Universal Robots PolyScope program: programa3.urp

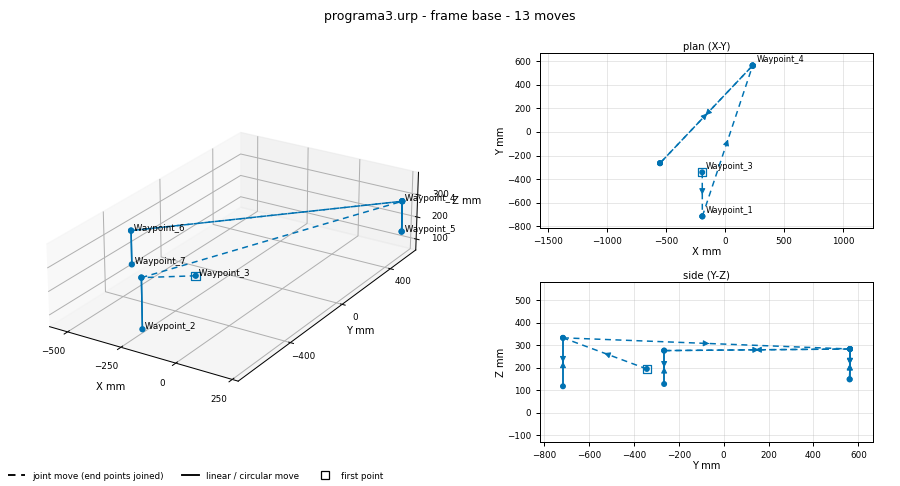
[picture p0: tool path of programa3.urp in frame base, 13 of 13 moves have a stored position in this frame; points joined in program order, loops and branches not executed]
Program programa3 (installation=default directory=/ursim/programs createdIn=5.26.1 lastSavedIn=5.26.1 robotSerialNumber=20195599999)
Calibrated DH parameters: a=[0, -0.425, -0.3922, 0, 0, 0]; d=[0.1625, 0, 0, 0.1333, 0.0997, 0.0996]; alpha=[1.570796, 0, 0, 1.570796, -1.570796, 0]; deltaTheta=[0, 0, 0, 0, 0, 0]
InitVariablesNode
Robot Program (runOnlyOnce=false)
  MoveJ speed 60 deg/s, acceleration 80 deg/s^2 (useActiveTCP=true optimoveEnabled=false optiMoveSpeed=0.3 optiMoveAcceleration=0.09) feature=Base
    Waypoint Waypoint_3: TCP in base x=-191.294 y=-341.962 z=194.296 mm, rx=-0.0012 ry=3.1163 rz=0.0389 rad; joints [-99.651, -91.23, -136.603, -43.818, 91.176, -9.713] deg; TCP offset x=0 y=0 z=0 mm, rx=0 ry=0 rz=0 rad
  Loop Forever
    MoveJ speed 60 deg/s, acceleration 80 deg/s^2 (useActiveTCP=true optimoveEnabled=false optiMoveSpeed=0.3 optiMoveAcceleration=0.09) feature=Base
      Waypoint Waypoint_1: TCP in base x=-190.469 y=-715.405 z=332.843 mm, rx=-0.0012 ry=3.1163 rz=0.0389 rad; joints [-94.715, -125.441, -65.388, -80.715, 91.313, -4.778] deg; TCP offset x=0 y=0 z=0 mm, rx=0 ry=0 rz=0 rad
    MoveL speed 250 mm/s, acceleration 1200 mm/s^2 (useActiveTCP=true optimoveEnabled=false optiMoveSpeed=0.3 optiMoveAcceleration=0.09) feature=Base
      Waypoint Waypoint_2: TCP in base x=-190.469 y=-715.405 z=116.996 mm, rx=-0.0012 ry=3.1163 rz=0.0389 rad; joints [-94.715, -137.604, -78.272, -55.669, 91.313, -4.778] deg; TCP offset x=0 y=0 z=0 mm, rx=0 ry=0 rz=0 rad
    Set DigitalOutput pin=digital_out[0]; digitalValue=1
    Wait Sleep waitTime=1
    MoveL speed 250 mm/s, acceleration 1200 mm/s^2 (useActiveTCP=true optimoveEnabled=false optiMoveSpeed=0.3 optiMoveAcceleration=0.09) feature=Base
      Waypoint Waypoint_1: TCP in base x=-190.469 y=-715.405 z=332.843 mm, rx=-0.0012 ry=3.1163 rz=0.0389 rad; joints [-94.715, -125.441, -65.388, -80.715, 91.313, -4.778] deg; TCP offset x=0 y=0 z=0 mm, rx=0 ry=0 rz=0 rad
    MoveJ speed 60 deg/s, acceleration 80 deg/s^2 (useActiveTCP=true optimoveEnabled=false optiMoveSpeed=0.3 optiMoveAcceleration=0.09) feature=Base
      Waypoint Waypoint_4: TCP in base x=235.914 y=562.656 z=283.122 mm, rx=2.8566 ry=-1.276 rz=-0.0517 rad; joints [79.536, -110.295, -96.699, -63.259, 92.011, 37.672] deg; TCP offset x=0 y=0 z=0 mm, rx=0 ry=0 rz=0 rad
    MoveL speed 250 mm/s, acceleration 1200 mm/s^2 (useActiveTCP=true optimoveEnabled=false optiMoveSpeed=0.3 optiMoveAcceleration=0.09) feature=Base
      Waypoint Waypoint_5: TCP in base x=238.855 y=560.992 z=148.209 mm, rx=2.8566 ry=-1.276 rz=-0.0517 rad; joints [79.229, -121.152, -103.988, -45.123, 92.01, 37.365] deg; TCP offset x=0 y=0 z=0 mm, rx=0 ry=0 rz=0 rad
    Set DigitalOutput pin=digital_out[0]; digitalValue=0
    Wait Sleep waitTime=1
    MoveL speed 250 mm/s, acceleration 1200 mm/s^2 (useActiveTCP=true optimoveEnabled=false optiMoveSpeed=0.3 optiMoveAcceleration=0.09) feature=Base
      Waypoint Waypoint_4: TCP in base x=235.914 y=562.656 z=283.122 mm, rx=2.8566 ry=-1.276 rz=-0.0517 rad; joints [79.536, -110.295, -96.699, -63.259, 92.011, 37.672] deg; TCP offset x=0 y=0 z=0 mm, rx=0 ry=0 rz=0 rad
    MoveJ speed 60 deg/s, acceleration 80 deg/s^2 (useActiveTCP=true optimoveEnabled=false optiMoveSpeed=0.3 optiMoveAcceleration=0.09) feature=Base
      Waypoint Waypoint_6: TCP in base x=-549.195 y=-264.968 z=275.959 mm, rx=2.1842 ry=2.2086 rz=0.0002 rad; joints [218.047, -110.703, -97.293, -62.267, 92.01, 37.405] deg; TCP offset x=0 y=0 z=0 mm, rx=0 ry=0 rz=0 rad
    MoveL speed 250 mm/s, acceleration 1200 mm/s^2 (useActiveTCP=true optimoveEnabled=false optiMoveSpeed=0.3 optiMoveAcceleration=0.09) feature=Base
      Waypoint Waypoint_7: TCP in base x=-549.195 y=-264.968 z=127.287 mm, rx=2.1842 ry=2.2086 rz=0.0002 rad; joints [218.047, -123.267, -104.538, -42.457, 92.01, 37.405] deg; TCP offset x=0 y=0 z=0 mm, rx=0 ry=0 rz=0 rad
    Set DigitalOutput pin=digital_out[0]; digitalValue=1
    Wait Sleep waitTime=1
    MoveL speed 250 mm/s, acceleration 1200 mm/s^2 (useActiveTCP=true optimoveEnabled=false optiMoveSpeed=0.3 optiMoveAcceleration=0.09) feature=Base
      Waypoint Waypoint_6: TCP in base x=-549.195 y=-264.968 z=275.959 mm, rx=2.1842 ry=2.2086 rz=0.0002 rad; joints [218.047, -110.703, -97.293, -62.267, 92.01, 37.405] deg; TCP offset x=0 y=0 z=0 mm, rx=0 ry=0 rz=0 rad
    MoveJ speed 60 deg/s, acceleration 80 deg/s^2 (useActiveTCP=true optimoveEnabled=false optiMoveSpeed=0.3 optiMoveAcceleration=0.09) feature=Base
      Waypoint Waypoint_4: TCP in base x=235.914 y=562.656 z=283.122 mm, rx=2.8566 ry=-1.276 rz=-0.0517 rad; joints [79.536, -110.295, -96.699, -63.259, 92.011, 37.672] deg; TCP offset x=0 y=0 z=0 mm, rx=0 ry=0 rz=0 rad
    MoveL speed 250 mm/s, acceleration 1200 mm/s^2 (useActiveTCP=true optimoveEnabled=false optiMoveSpeed=0.3 optiMoveAcceleration=0.09) feature=Base
      Waypoint Waypoint_5: TCP in base x=238.855 y=560.992 z=148.209 mm, rx=2.8566 ry=-1.276 rz=-0.0517 rad; joints [79.229, -121.152, -103.988, -45.123, 92.01, 37.365] deg; TCP offset x=0 y=0 z=0 mm, rx=0 ry=0 rz=0 rad
    Set DigitalOutput pin=digital_out[0]; digitalValue=0
    Wait Sleep waitTime=1
    MoveL speed 250 mm/s, acceleration 1200 mm/s^2 (useActiveTCP=true optimoveEnabled=false optiMoveSpeed=0.3 optiMoveAcceleration=0.09) feature=Base
      Waypoint Waypoint_4: TCP in base x=235.914 y=562.656 z=283.122 mm, rx=2.8566 ry=-1.276 rz=-0.0517 rad; joints [79.536, -110.295, -96.699, -63.259, 92.011, 37.672] deg; TCP offset x=0 y=0 z=0 mm, rx=0 ry=0 rz=0 rad
    Wait DigitalInput pin=digital_in[0]; digitalValue=1
